(* Logix 5000 project; controller cow Emulate 5570 rev 36.11; software revision 36.00 *)

TASK MainTask (continuous, watchdog 500 ms) : MainProgram, Recipe, LED_UDP

MODULES
   Local : Emulate 5570 (ICP 0, rev 36.11)
      EN2T : 1756-EN2T (ICP 1, rev 12.1)
         Cow : 1756-ENBT (Ethernet 192.168.1.1, rev 5.1, Output RPI 10 ms)
            Caw1 : vendor 1 type 0 code 15 (ICP 0, rev 1.1, Output RPI 20 ms)
END_MODULES

TYPE ActLog :
STRUCT
   Time : DINT;
   STS : INT;
END_STRUCT
END_TYPE

TYPE Batch :
STRUCT
   Clear_Data : BOOL;
   LL : BOOL;
   Report_Log : BOOL;
   Value : INT;
   Batch : INT;
   Fall : INT;
   Target : INT;
   Net_Gross : DINT;
   Report : DINT[7];
   Scale : SCALE_WEIGHT;
   BinLog : BinLog[20];
END_STRUCT
END_TYPE

TYPE BinLog :
STRUCT
   SourceBin : INT;
   DestBin : INT;
   SetWeight : INT;
   StartTime : DINT;
   StopTime : DINT;
   pNumber : DINT;
   pNumberS : DINT[2];
END_STRUCT
END_TYPE

TYPE DateTime_Type :
STRUCT
   Year : DINT;
   Month : DINT;
   Day : DINT;
   Hour : DINT;
   Minute : DINT;
   Second : DINT;
   Microseconds : DINT;
END_STRUCT
END_TYPE

TYPE Part_Manual_Type :
STRUCT
   Bin : INT[5];
   Number : DINT[10];
   SetWeight : REAL[5];
   RealWeight : REAL[5];
   ErrorWeight : REAL[5];
END_STRUCT
END_TYPE

TYPE Part_Type :
STRUCT
   Bin : INT[20];
   Bin_Index : INT[20];
   Number : DINT[20];
   SetWeight : REAL[20];
   RealWeight : REAL[20];
   ErrorWeight : REAL[20];
END_STRUCT
END_TYPE

TYPE Part_Type_Hand :
STRUCT
   Number : DINT[30];
   SetWeight : REAL[30];
   RealWeight : REAL[30];
   ErrorWeight : REAL[30];
END_STRUCT
END_TYPE

TYPE Recipe_Type :
STRUCT
   Number : DINT[3];
   Desc : DINT[8];
   BatchSet : DINT;
   Date : DINT;
   pNumber : DINT[20];
   pSetWeight : REAL[20];
END_STRUCT
END_TYPE

TYPE REQUEST_PARAMETERS :
STRUCT
   Type : DINT;
   Addr : SockAddr;
END_STRUCT
END_TYPE

TYPE ScheduleLog :
STRUCT
   Number : DINT[3];
   StartTime : DINT;
   Batch : DINT;
END_STRUCT
END_TYPE

TYPE SockAddr :
STRUCT
   Family : INT;
   Port : INT;
   Addr : DINT;
END_STRUCT
END_TYPE

TYPE STR_OUT :
STRUCT
   LEN : DINT;
   BUFF : SINT[480];
END_STRUCT
END_TYPE

TYPE String20 :
STRUCT
   LEN : DINT;
   DATA : SINT[20];
END_STRUCT
END_TYPE

TYPE Sys_Data :
STRUCT
   MC : BOOL;
   AUTO_START : BOOL;
   AUTO_STOP : BOOL;
   EM : BOOL;
   AUTO : BOOL;
   MANUAL : BOOL;
   SIMULATE : BOOL;
   Monitor_PLC5 : BOOL;
   FlashFast : BOOL;
   FlashSlow : BOOL;
   Err_Reset : BOOL;
   PB : BOOL;
   Power : BOOL;
   Auto_Start_Enable : BOOL;
   Change_Bin_Ack : BOOL;
   FA : BOOL;
   Bin_Num_OK : BOOL;
   ClearLog : BOOL;
   Flag : BOOL;
   Alarm : BOOL;
   Compare_Bin : BOOL;
   OK : BOOL;
   BinLogStart : BOOL;
   Report_Log : BOOL;
   DropStop : BOOL;
   DM : BOOL;
   DropTimeS : INT;
   DropTime : TON_Second;
   BIN_SEL : INT;
   BIN_PLC : INT;
   BIN_SEL1 : INT;
   BinS_SEL1 : INT;
   BinS_SEL : INT;
   Day : INT;
   Day_Hour : INT;
   Year : INT;
   START_ACC : INT;
   Stop_ACC : INT;
   SEL_BIN : INT;
   MSG_ID : INT;
   MMDDHHMMS : DINT;
   sNumber : DINT;
   pNumber : DINT;
   NumberS : DINT[2];
   NumberSel : DINT[2];
   ActLog : ActLog[20];
   ChangeBin : TON_Second;
   StartT : TON_Second;
   StopT : TON_Second;
   TimeSet : TON_Second;
   SeqStartT : INT[21];
   SeqStopT : INT[21];
   BinLog : BinLog[20];
   SEL_Weight : REAL;
   Report : DINT[7];
END_STRUCT
END_TYPE

TYPE System_Common :
STRUCT
   Simulate : BOOL;
   Monitor_PLC5 : BOOL;
   FlashFast : BOOL;
   FlashSlow : BOOL;
   SY_PW_OK : BOOL;
   Err_Reset : BOOL;
   ClearLog : BOOL;
   PSH : BOOL;
   PSL : BOOL;
   Air_CLEAR : BOOL;
   DAY : INT;
   Day_Hour : INT;
   Year : INT;
   MMDDHHMMs : DINT;
END_STRUCT
END_TYPE

TYPE WRT_DATA :
STRUCT
   Timeout : DINT;
   ToAddr : SockAddr;
   Buffer : STR_OUT;
END_STRUCT
END_TYPE

ADD_ON_INSTRUCTION Air_Hammer   (* revision 1.0 *)
// 氣槌
VAR_INPUT
   PBM : BOOL; {visible}   // On/Off開關
   PB : BOOL;
   AB : BOOL;
   TH : BOOL;
END_VAR
VAR_OUTPUT
   SV : BOOL; {access Read Only, visible}   // 運轉
   MC : BOOL; {access Read Only}
   GL : BOOL; {access Read Only, visible}   // 運轉指示
END_VAR
VAR_INPUT
   Auto_on : BOOL; {visible}   // 連續
END_VAR
VAR_OUTPUT
   MotorType : BOOL; {visible}
END_VAR
VAR_IN_OUT
   Sys : Sys_Data; {required}   // 系統設定
END_VAR
VAR
   ONS : DINT; {access None}
   On_Time : TIMER := (PRE := 2000); {access None}
   Repeat_T : TIMER := (PRE := 2000); {access None}
END_VAR

ROUTINE Logic   (* ladder *)
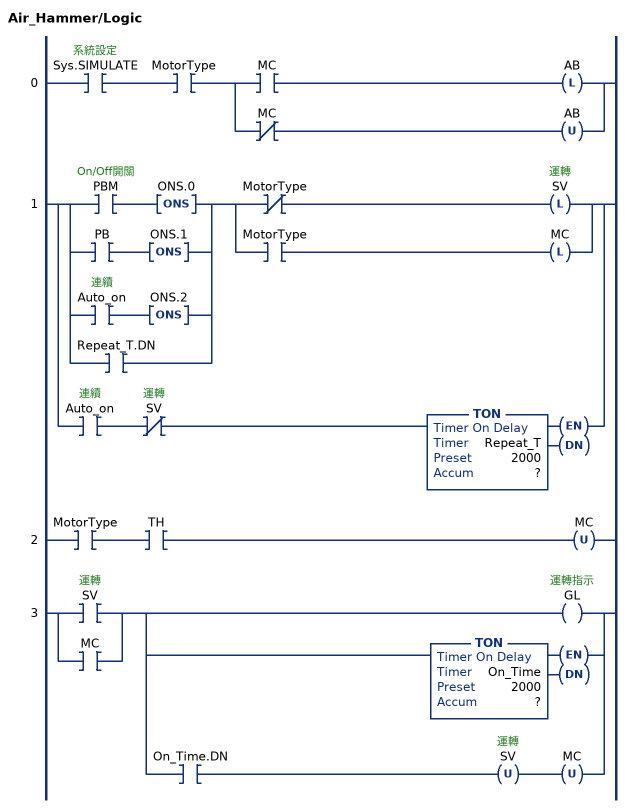
   0: XIC(Sys.SIMULATE)XIC(MotorType)[XIC(MC) OTL(AB) ,XIO(MC) OTU(AB) ];
   1: [[XIC(PBM) ONS(ONS.0) ,XIC(PB) ONS(ONS.1) ,XIC(Auto_on) ONS(ONS.2) ,XIC(Repeat_T.DN) ] [XIO(MotorType) OTL(SV) ,XIC(MotorType) OTL(MC) ] ,XIC(Auto_on) XIO(SV) TON(Repeat_T,?,?) ];
   2: XIC(MotorType)XIC(TH)OTU(MC);
   3: [XIC(SV) ,XIC(MC) ][OTE(GL) ,TON(On_Time,?,?) ,XIC(On_Time.DN) OTU(SV) OTU(MC) ];
END_ROUTINE
END_ADD_ON_INSTRUCTION

ADD_ON_INSTRUCTION Bin_Raw   (* revision 1.0 *)
VAR_OUTPUT
   HL : BOOL; {visible}
   LL : BOOL; {visible}
   FA : BOOL; {access Read Only, visible}
   Bin_sel : BOOL;
   Bin_Sel_OK : BOOL; {access Read Only}
   BIN_SELECTED : BOOL; {access Read Only}
   BIN_SELECTED1 : BOOL; {access Read Only}
   YL : BOOL; {access Read Only, visible}
   SV : BOOL;
END_VAR
VAR_INPUT
   LSO : BOOL;
END_VAR
VAR_OUTPUT
   CMD : BOOL; {visible}
   HGL : BOOL; {access Read Only, visible}
END_VAR
VAR_INPUT
   LS : BOOL; {access Read Only, visible}
   Change_Bin_Ack : BOOL;
   Bin_sel_No : BOOL;
END_VAR
VAR_OUTPUT
   HiSpeed : BOOL; {visible}
   LowSpeed : BOOL; {visible}
   DM : BOOL; {access Read Only, visible}
   SV_ON : BOOL;
   Disable : BOOL; {visible}
END_VAR
VAR_INPUT
   PB : BOOL;
END_VAR
VAR_OUTPUT
   GL : BOOL;
   Local_Sel : BOOL;
END_VAR
VAR_INPUT
   Bin : INT; {visible}
   Bin_ID : INT; {access Read Only, visible}
   Fall : REAL; {visible}
   Hi_Speed : INT := 80; {visible}
   Low_Speed : INT := 20; {visible}
   Low_Weight : INT := 5; {visible}
   Number : DINT; {visible}
   N0 : ALIAS FOR NumberS[0]; {visible}
   N1 : ALIAS FOR NumberS[1]; {visible}
END_VAR
VAR_IN_OUT
   Sys : Sys_Data; {required}
END_VAR
VAR
   Timer : TIMER := (PRE := 4000); {access None}
   ons : DINT; {access None}
   LVH_DELAY : TIMER := (PRE := 2000); {access None}
   NumberS : DINT[2];
END_VAR

ROUTINE Logic   (* ladder *)
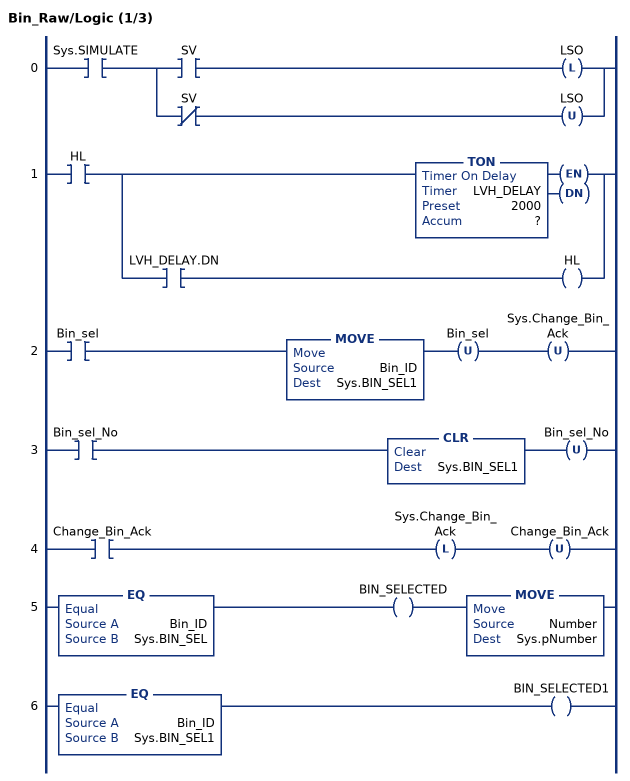
   0: XIC(Sys.SIMULATE)[XIC(SV) OTL(LSO) ,XIO(SV) OTU(LSO) ];
   1: XIC(HL)[TON(LVH_DELAY,?,?) ,XIC(LVH_DELAY.DN) OTE(HL) ];
   2: XIC(Bin_sel)MOVE(Bin_ID,Sys.BIN_SEL1)OTU(Bin_sel)OTU(Sys.Change_Bin_Ack);
   3: XIC(Bin_sel_No)CLR(Sys.BIN_SEL1)OTU(Bin_sel_No);
   4: XIC(Change_Bin_Ack)OTL(Sys.Change_Bin_Ack)OTU(Change_Bin_Ack);
   5: EQ(Bin_ID,Sys.BIN_SEL)OTE(BIN_SELECTED)MOVE(Number,Sys.pNumber);
   6: EQ(Bin_ID,Sys.BIN_SEL1)OTE(BIN_SELECTED1);
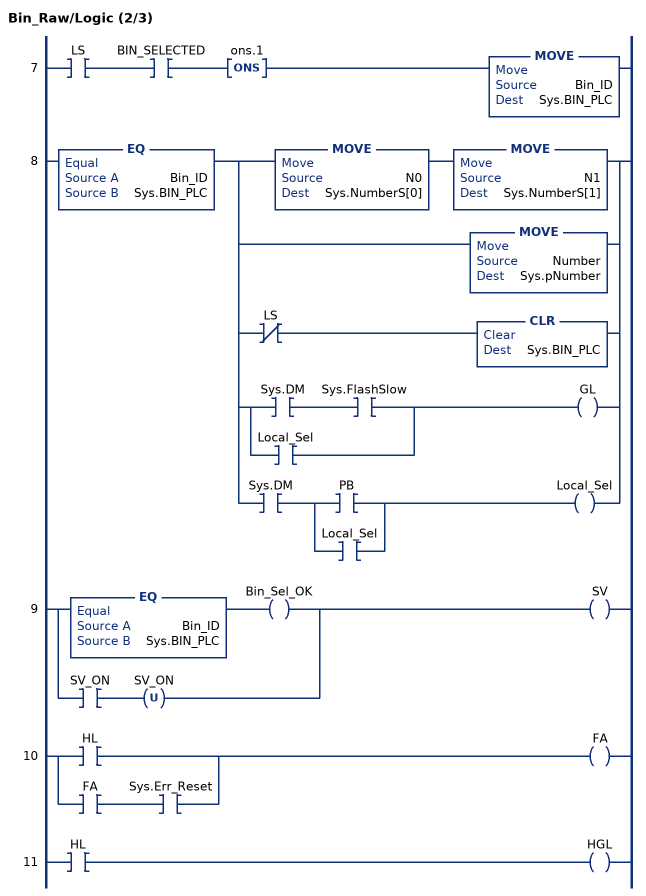
   7: XIC(LS)XIC(BIN_SELECTED)ONS(ons.1)MOVE(Bin_ID,Sys.BIN_PLC);
   8: EQ(Bin_ID,Sys.BIN_PLC)[MOVE(N0,Sys.NumberS[0]) MOVE(N1,Sys.NumberS[1]) ,MOVE(Number,Sys.pNumber) ,XIO(LS) CLR(Sys.BIN_PLC) ,[XIC(Sys.DM) XIC(Sys.FlashSlow) ,XIC(Local_Sel) ] OTE(GL) ,XIC(Sys.DM) [XIC(PB) ,XIC(Local_Sel) ] OTE(Local_Sel) ];
   9: [EQ(Bin_ID,Sys.BIN_PLC) OTE(Bin_Sel_OK) ,XIC(SV_ON) OTU(SV_ON) ]OTE(SV);
   10: [XIC(HL) ,XIC(FA) XIC(Sys.Err_Reset) ]OTE(FA);
   11: XIC(HL)OTE(HGL);
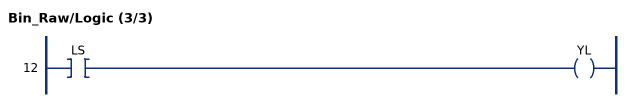
   12: XIC(LS)OTE(YL);
END_ROUTINE
END_ADD_ON_INSTRUCTION

ADD_ON_INSTRUCTION Branch_SV2   (* revision 1.0 *)
VAR_INPUT
   LSY : BOOL; {visible}
   LSX : BOOL; {visible}
END_VAR
VAR_OUTPUT
   SVX : BOOL; {access Read Only, visible}
   SVY : BOOL; {access Read Only, visible}
   FA : BOOL; {visible}
   GLX : BOOL; {access Read Only}
   GLY : BOOL; {access Read Only}
   Manual : BOOL;
   SVXPB : BOOL; {visible}
   SVYPB : BOOL; {visible}
   Auto : BOOL;
   Not_AOI_Control : BOOL; {visible}
END_VAR
VAR_INPUT
   InterLock : BOOL;
END_VAR
VAR_IN_OUT
   STS : INT; {required}
   Sys : Sys_Data; {required}
END_VAR
VAR
   SV : BOOL; {access None}
   ONS : DINT; {access None}
   DELAY : TIMER := (PRE := 3000); {access None}
   ActLog : ActLog[20];
   LastOnTime : DINT;
   LastOffTime : DINT;
END_VAR

ROUTINE Logic   (* ladder *)
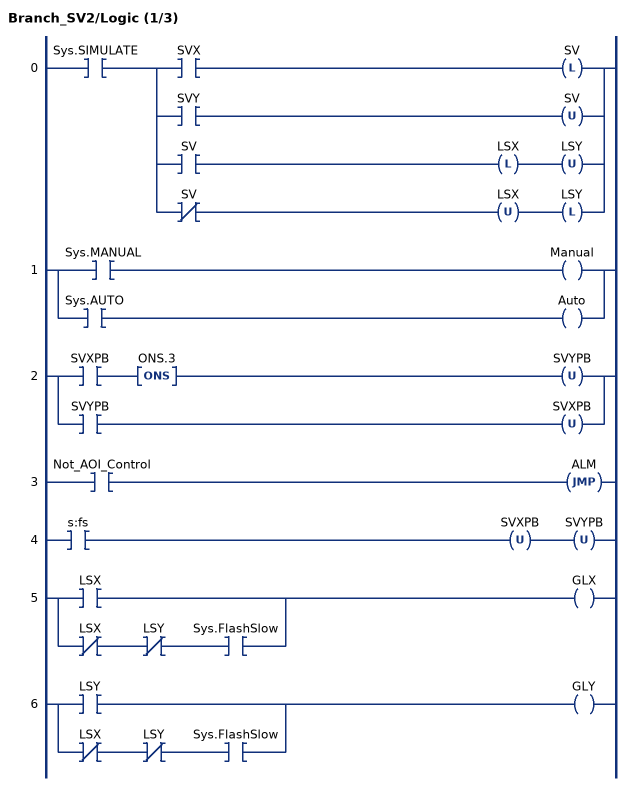
   0: XIC(Sys.SIMULATE)[XIC(SVX) OTL(SV) ,XIC(SVY) OTU(SV) ,XIC(SV) OTL(LSX) OTU(LSY) ,XIO(SV) OTU(LSX) OTL(LSY) ];
   1: [XIC(Sys.MANUAL) OTE(Manual) ,XIC(Sys.AUTO) OTE(Auto) ];
   2: [XIC(SVXPB) ONS(ONS.3) OTU(SVYPB) ,XIC(SVYPB) OTU(SVXPB) ];
   3: XIC(Not_AOI_Control)JMP(ALM);
   4: XIC(s:fs)OTU(SVXPB)OTU(SVYPB);
   5: [XIC(LSX) ,XIO(LSX) XIO(LSY) XIC(Sys.FlashSlow) ]OTE(GLX);
   6: [XIC(LSY) ,XIO(LSX) XIO(LSY) XIC(Sys.FlashSlow) ]OTE(GLY);
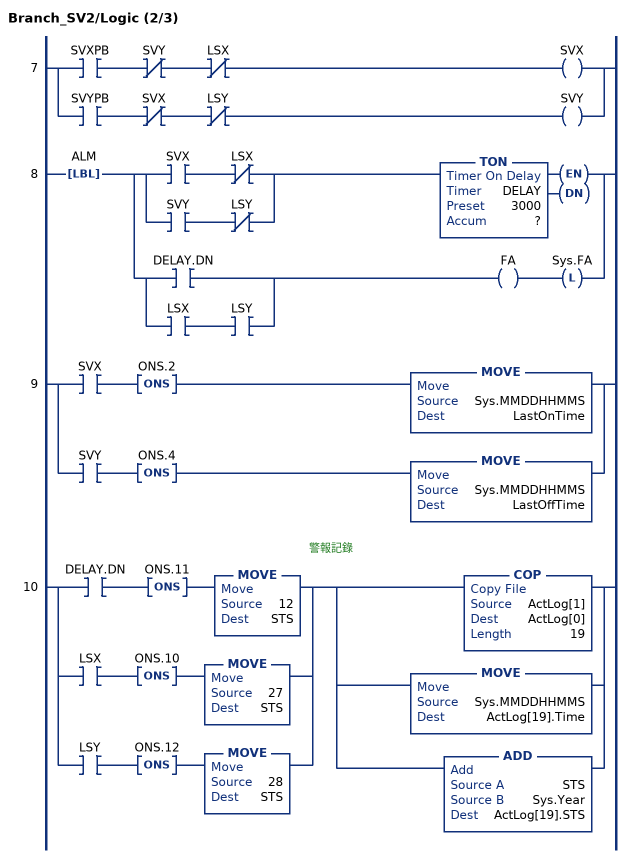
   7: [XIC(SVXPB) XIO(SVY) XIO(LSX) OTE(SVX) ,XIC(SVYPB) XIO(SVX) XIO(LSY) OTE(SVY) ];
   8: LBL(ALM)[[XIC(SVX) XIO(LSX) ,XIC(SVY) XIO(LSY) ] TON(DELAY,?,?) ,[XIC(DELAY.DN) ,XIC(LSX) XIC(LSY) ] OTE(FA) OTL(Sys.FA) ];
   9: [XIC(SVX) ONS(ONS.2) MOVE(Sys.MMDDHHMMS,LastOnTime) ,XIC(SVY) ONS(ONS.4) MOVE(Sys.MMDDHHMMS,LastOffTime) ];
   // 警報記錄
   10: [XIC(DELAY.DN) ONS(ONS.11) MOVE(12,STS) ,[XIC(LSX) ONS(ONS.10) MOVE(27,STS) ,XIC(LSY) ONS(ONS.12) MOVE(28,STS) ] ][COP(ActLog[1],ActLog[0],19) ,MOVE(Sys.MMDDHHMMS,ActLog[19].Time) ,ADD(STS,Sys.Year,ActLog[19].STS) ];
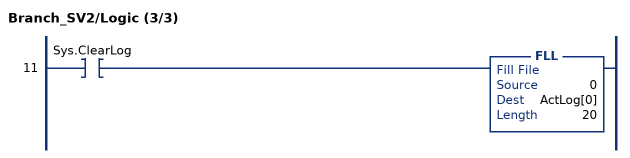
   11: XIC(Sys.ClearLog)FLL(0,ActLog[0],20);
END_ROUTINE
END_ADD_ON_INSTRUCTION

ADD_ON_INSTRUCTION DateTime_String   (* revision 1.0 *)
VAR_IN_OUT
   Now : DateTime_Type; {required}
   DateTimes : STRING; {required}
END_VAR
VAR
   HOUR : STRING; {access None}
   MINUTE : STRING; {access None}
   SECOND : STRING; {access None}
   zero : STRING := '0'; {access None}
   COLN : STRING := ':'; {access None}
   Prev_Second : DINT; {access None}
   Day : STRING; {access None}
   Month : STRING; {access None}
   Year : STRING; {access None}
   Da : STRING := '/'; {access None}
   Blank : STRING := '  '; {access None}
END_VAR

ROUTINE Logic   (* ladder *)
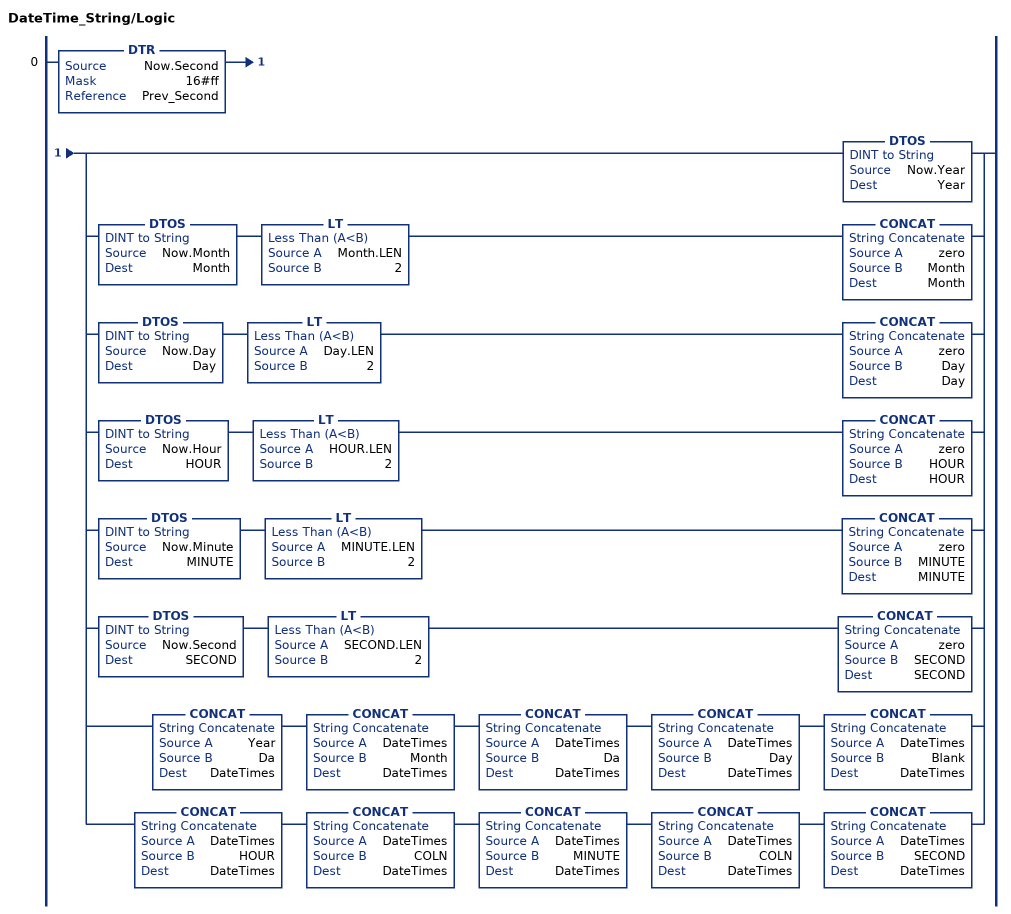
   0: DTR(Now.Second,16#ff,Prev_Second)[DTOS(Now.Year,Year) ,DTOS(Now.Month,Month) LT(Month.LEN,2) CONCAT(zero,Month,Month) ,DTOS(Now.Day,Day) LT(Day.LEN,2) CONCAT(zero,Day,Day) ,DTOS(Now.Hour,HOUR) LT(HOUR.LEN,2) CONCAT(zero,HOUR,HOUR) ,DTOS(Now.Minute,MINUTE) LT(MINUTE.LEN,2) CONCAT(zero,MINUTE,MINUTE) ,DTOS(Now.Second,SECOND) LT(SECOND.LEN,2) CONCAT(zero,SECOND,SECOND) ,CONCAT(Year,Da,DateTimes) CONCAT(DateTimes,Month,DateTimes) CONCAT(DateTimes,Da,DateTimes) CONCAT(DateTimes,Day,DateTimes) CONCAT(DateTimes,Blank,DateTimes) ,CONCAT(DateTimes,HOUR,DateTimes) CONCAT(DateTimes,COLN,DateTimes) CONCAT(DateTimes,MINUTE,DateTimes) CONCAT(DateTimes,COLN,DateTimes) CONCAT(DateTimes,SECOND,DateTimes) ];
END_ROUTINE
END_ADD_ON_INSTRUCTION

ADD_ON_INSTRUCTION Divider   (* revision 1.0 *)
VAR_INPUT
   AB : BOOL; {visible}
END_VAR
VAR_OUTPUT
   MC : BOOL; {access Read Only, visible}
END_VAR
VAR_INPUT
   TH : BOOL; {visible}
END_VAR
VAR_OUTPUT
   FA : BOOL; {visible}
END_VAR
VAR_INPUT
   MANUAL_ON : BOOL; {visible}
   AUTO_ON : BOOL;
END_VAR
VAR_OUTPUT
   MANUAL : BOOL; {visible}
   OverTime : BOOL; {visible}
   LS1 : ALIAS FOR LS.1;
   LS2 : ALIAS FOR LS.2;
   LS3 : ALIAS FOR LS.3;
   LS4 : ALIAS FOR LS.4;
   LS5 : ALIAS FOR LS.5;
   LS6 : ALIAS FOR LS.6;
   LS7 : ALIAS FOR LS.7;
   LS8 : ALIAS FOR LS.8;
   LS9 : ALIAS FOR LS.9;
   LS10 : ALIAS FOR LS.10;
   LS11 : ALIAS FOR LS.11;
   LS12 : ALIAS FOR LS.12;
   LS_ON : BOOL;
   Not_AOI_Control : BOOL; {visible}
   Bin_select : BOOL; {visible}
   Simulate : ALIAS FOR Simulate_POS.ACC; {access Read Only}
END_VAR
VAR_IN_OUT
   STS : INT; {required}
   Sys : Sys_Data; {required}
END_VAR
VAR
   DELAY : TIMER := (PRE := 1000); {access None}
   Simulate_TIMER : TIMER := (PRE := 1000); {access None}
   Simulate_POS : COUNTER := (PRE := 7); {access Read Only}
   ONS : DINT; {access None}
   error_delay : TIMER := (PRE := 5000); {access None}
   MC_RUN_T : TIMER := (PRE := 40000); {access None}
   LS : DINT;
   ActLog : ActLog[20];
   LastOnTime : DINT;
   LastOffTime : DINT;
END_VAR

ROUTINE Logic   (* ladder *)
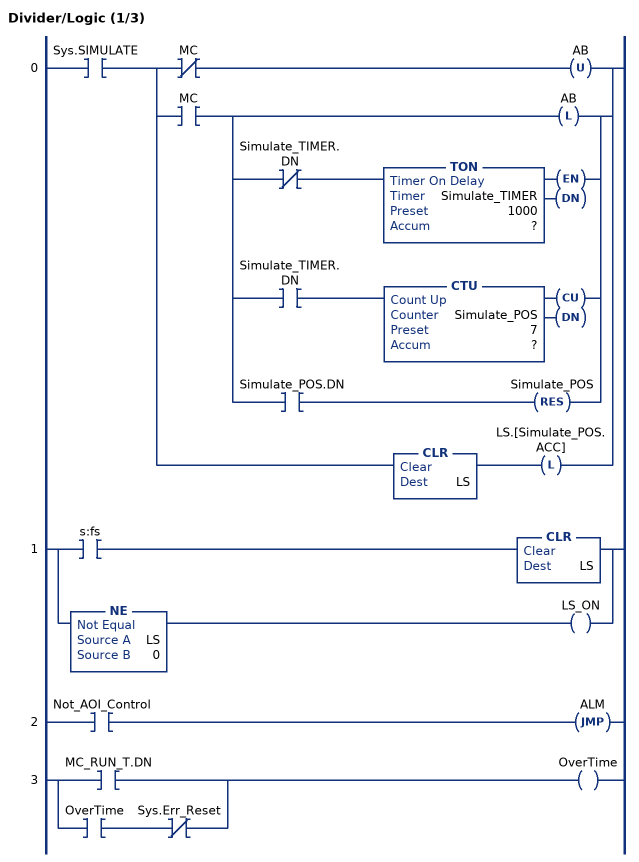
   0: XIC(Sys.SIMULATE)[XIO(MC) OTU(AB) ,XIC(MC) [OTL(AB) ,XIO(Simulate_TIMER.DN) TON(Simulate_TIMER,?,?) ,XIC(Simulate_TIMER.DN) CTU(Simulate_POS,?,?) ,XIC(Simulate_POS.DN) RES(Simulate_POS) ] ,CLR(LS) OTL(LS.[Simulate_POS.ACC]) ];
   1: [XIC(s:fs) CLR(LS) ,NE(LS,0) OTE(LS_ON) ];
   2: XIC(Not_AOI_Control)JMP(ALM);
   3: [XIC(MC_RUN_T.DN) ,XIC(OverTime) XIO(Sys.Err_Reset) ]OTE(OverTime);
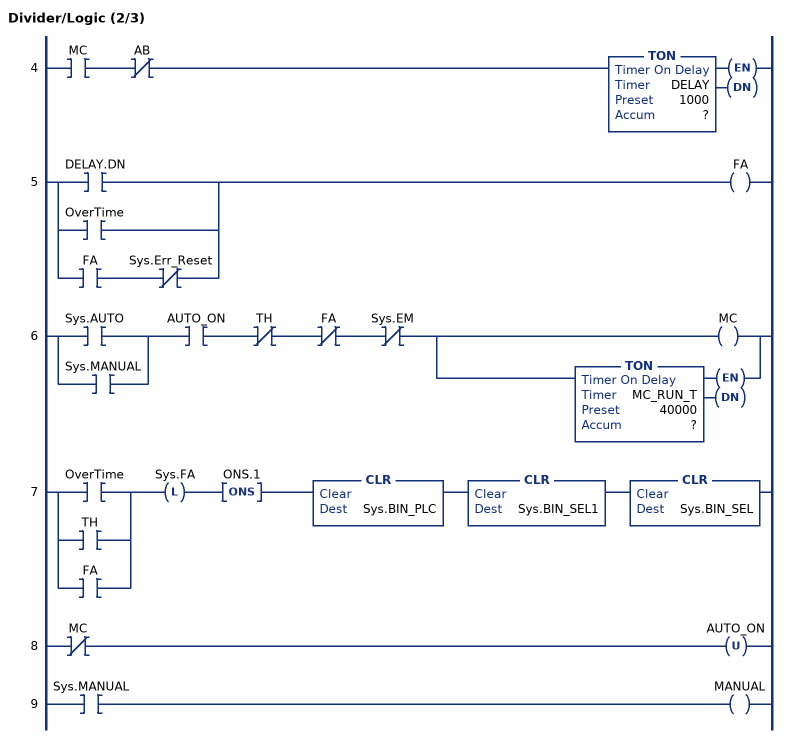
   4: XIC(MC)XIO(AB)TON(DELAY,?,?);
   5: [XIC(DELAY.DN) ,XIC(OverTime) ,XIC(FA) XIO(Sys.Err_Reset) ]OTE(FA);
   6: [XIC(Sys.AUTO) ,XIC(Sys.MANUAL) ]XIC(AUTO_ON)XIO(TH)XIO(FA)XIO(Sys.EM)[OTE(MC) ,TON(MC_RUN_T,?,?) ];
   7: [XIC(OverTime) ,XIC(TH) ,XIC(FA) ]OTL(Sys.FA)ONS(ONS.1)CLR(Sys.BIN_PLC)CLR(Sys.BIN_SEL1)CLR(Sys.BIN_SEL);
   8: XIO(MC)OTU(AUTO_ON);
   9: XIC(Sys.MANUAL)OTE(MANUAL);
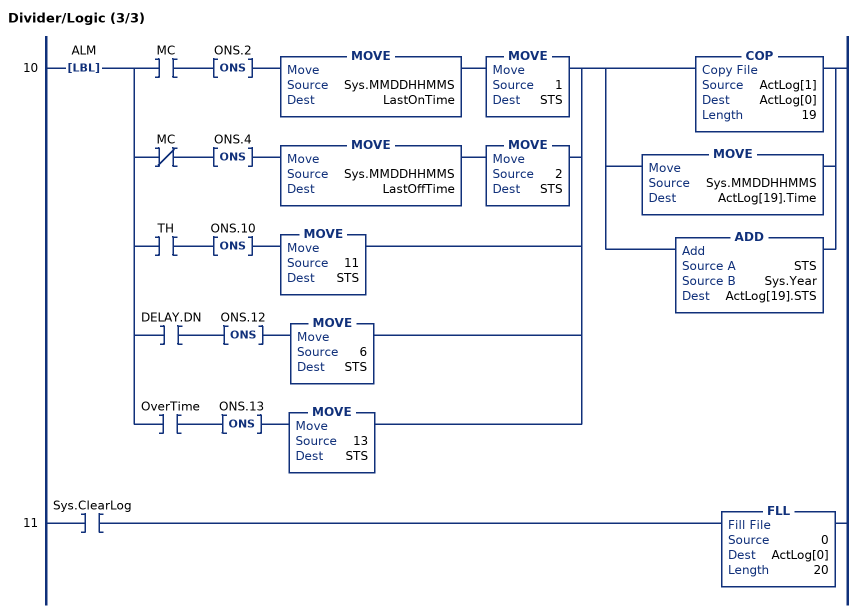
   10: LBL(ALM)[XIC(MC) ONS(ONS.2) MOVE(Sys.MMDDHHMMS,LastOnTime) MOVE(1,STS) ,XIO(MC) ONS(ONS.4) MOVE(Sys.MMDDHHMMS,LastOffTime) MOVE(2,STS) ,XIC(TH) ONS(ONS.10) MOVE(11,STS) ,XIC(DELAY.DN) ONS(ONS.12) MOVE(6,STS) ,XIC(OverTime) ONS(ONS.13) MOVE(13,STS) ][COP(ActLog[1],ActLog[0],19) ,MOVE(Sys.MMDDHHMMS,ActLog[19].Time) ,ADD(STS,Sys.Year,ActLog[19].STS) ];
   11: XIC(Sys.ClearLog)FLL(0,ActLog[0],20);
END_ROUTINE
END_ADD_ON_INSTRUCTION

ADD_ON_INSTRUCTION Gate   (* revision 1.0 *)
VAR_INPUT
   LSO : BOOL; {visible}
   LSK : BOOL; {visible}
END_VAR
VAR_OUTPUT
   SV : BOOL; {visible}
   Auto_On : BOOL;
   Manual : BOOL; {visible}
   FA : BOOL; {visible}
   OPEN : BOOL; {visible}
   InterLock : BOOL; {access Read Only, visible}
   Auto : BOOL;
   PB : BOOL;
   GL : BOOL; {access Read Only, visible}
END_VAR
VAR_INPUT
   LL : BOOL;
END_VAR
VAR_OUTPUT
   Not_AOI_Control : BOOL; {visible}
   Lock : BOOL;
   LSO_Delay : BOOL;
   Off_Delay : BOOL;
END_VAR
VAR_IN_OUT
   STS : INT; {required}
   Sys : Sys_Data; {required}
END_VAR
VAR
   Open_Delay : TIMER := (PRE := 500); {access None}
   Close_Delay : TIMER := (PRE := 500); {access None}
   TimeOut : TIMER := (PRE := 3000); {access None}
   Interlock_Delay : TIMER := (PRE := 500); {access None}
   ActLog : ActLog[20];
   ONS : DINT; {access None}
   LS_Delay : TIMER[2] := ([0].PRE := 1000, [1].PRE := 1000); {access None}
   PB_Delay : TIMER := (PRE := 500); {access None}
   LSO_DelayT : TIMER := (PRE := 2000); {access None}
   off_DelayT : TIMER := (PRE := 2000); {access None}
END_VAR

ROUTINE Logic   (* ladder *)
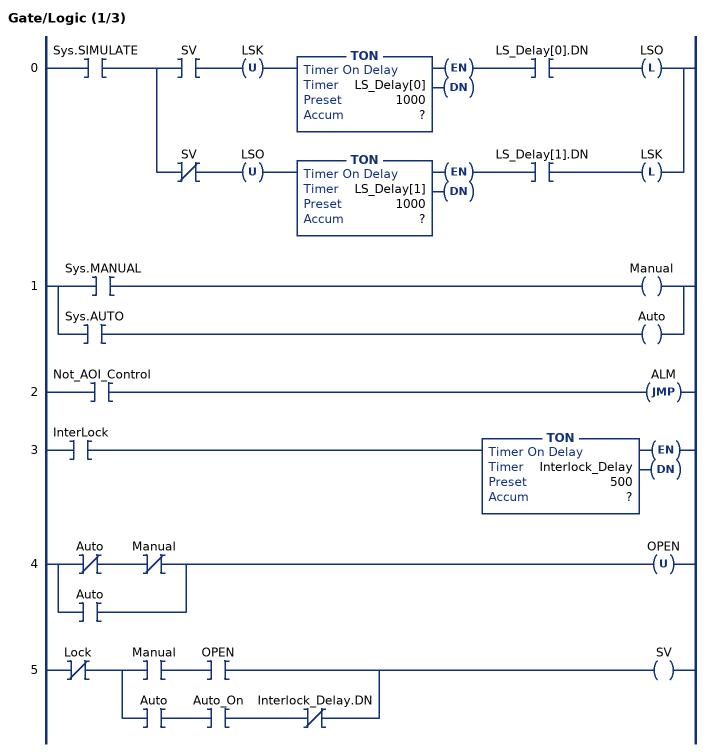
   0: XIC(Sys.SIMULATE)[XIC(SV) OTU(LSK) TON(LS_Delay[0],?,?) XIC(LS_Delay[0].DN) OTL(LSO) ,XIO(SV) OTU(LSO) TON(LS_Delay[1],?,?) XIC(LS_Delay[1].DN) OTL(LSK) ];
   1: [XIC(Sys.MANUAL) OTE(Manual) ,XIC(Sys.AUTO) OTE(Auto) ];
   2: XIC(Not_AOI_Control)JMP(ALM);
   3: XIC(InterLock)TON(Interlock_Delay,?,?);
   4: [XIO(Auto) XIO(Manual) ,XIC(Auto) ]OTU(OPEN);
   5: XIO(Lock)[XIC(Manual) XIC(OPEN) ,XIC(Auto) XIC(Auto_On) XIO(Interlock_Delay.DN) ]OTE(SV);
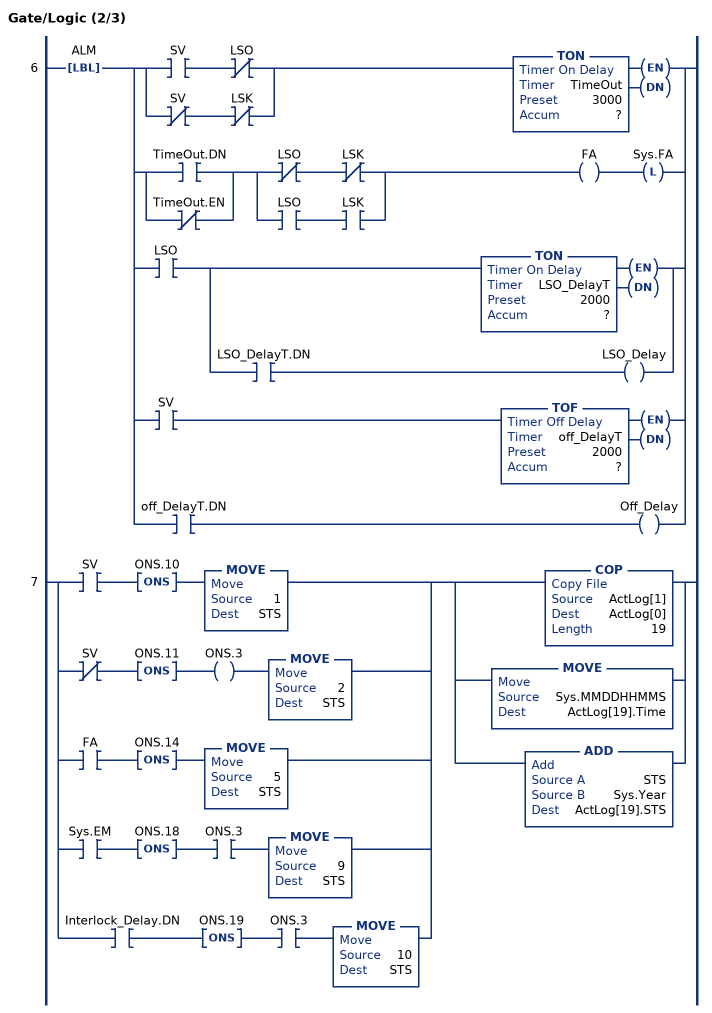
   6: LBL(ALM)[[XIC(SV) XIO(LSO) ,XIO(SV) XIO(LSK) ] TON(TimeOut,?,?) ,[XIC(TimeOut.DN) ,XIO(TimeOut.EN) ] [XIO(LSO) XIO(LSK) ,XIC(LSO) XIC(LSK) ] OTE(FA) OTL(Sys.FA) ,XIC(LSO) [TON(LSO_DelayT,?,?) ,XIC(LSO_DelayT.DN) OTE(LSO_Delay) ] ,XIC(SV) TOF(off_DelayT,?,?) ,XIC(off_DelayT.DN) OTE(Off_Delay) ];
   7: [[XIC(SV) ONS(ONS.10) MOVE(1,STS) ,XIO(SV) ONS(ONS.11) OTE(ONS.3) MOVE(2,STS) ] ,XIC(FA) ONS(ONS.14) MOVE(5,STS) ,XIC(Sys.EM) ONS(ONS.18) XIC(ONS.3) MOVE(9,STS) ,XIC(Interlock_Delay.DN) ONS(ONS.19) XIC(ONS.3) MOVE(10,STS) ][COP(ActLog[1],ActLog[0],19) ,MOVE(Sys.MMDDHHMMS,ActLog[19].Time) ,ADD(STS,Sys.Year,ActLog[19].STS) ];
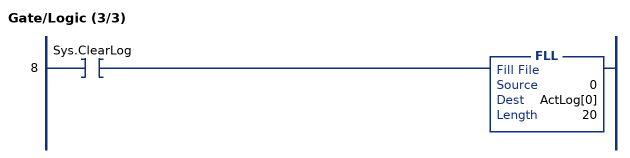
   8: XIC(Sys.ClearLog)FLL(0,ActLog[0],20);
END_ROUTINE
END_ADD_ON_INSTRUCTION

ADD_ON_INSTRUCTION Inverter   (* revision 1.0 *)
VAR_INPUT
   AB : BOOL; {visible}
END_VAR
VAR_OUTPUT
   MC : BOOL; {access Read Only, visible}
END_VAR
VAR_INPUT
   TH : BOOL; {visible}
END_VAR
VAR_OUTPUT
   RMC : BOOL; {visible}
   AUTO_ON : BOOL;
END_VAR
VAR_INPUT
   Manual_HZ : INT := 10; {visible}
   HZ : INT; {visible}
END_VAR
VAR_IN_OUT
   STS : INT; {required}
   Sys : Sys_Data; {required}
END_VAR
VAR
   DELAY : TIMER := (PRE := 100); {access None}
   ONS : DINT; {access None}
   AlmLog : DINT[6]; {access Read Only}
   ALM_ID : DINT; {access None}
   RunTIme : TIMER := (PRE := 99999); {access Read Only}
END_VAR

ROUTINE Logic   (* ladder *)
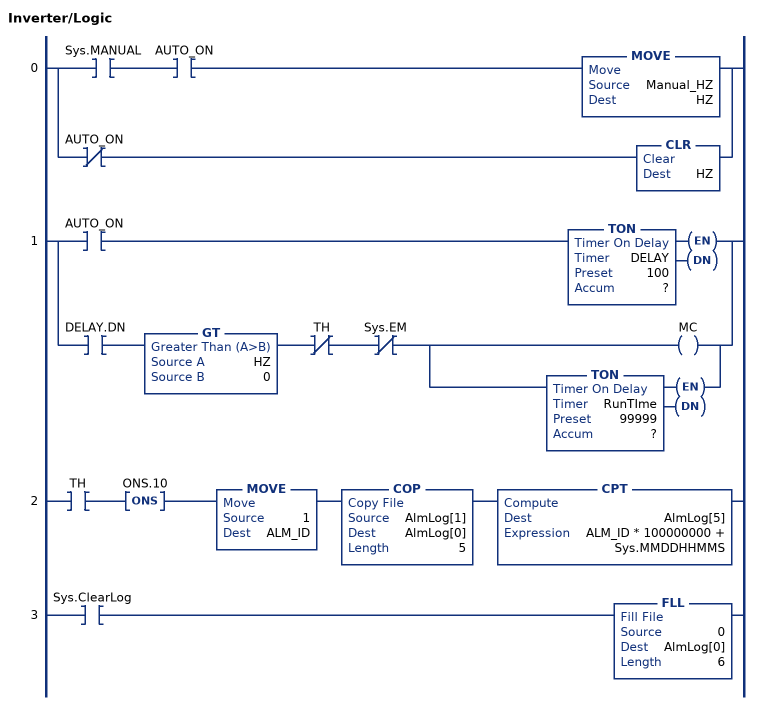
   0: [XIC(Sys.MANUAL) XIC(AUTO_ON) MOVE(Manual_HZ,HZ) ,XIO(AUTO_ON) CLR(HZ) ];
   1: [XIC(AUTO_ON) TON(DELAY,?,?) ,XIC(DELAY.DN) GT(HZ,0) XIO(TH) XIO(Sys.EM) [OTE(MC) ,TON(RunTIme,?,?) ] ];
   2: XIC(TH)ONS(ONS.10)MOVE(1,ALM_ID)COP(AlmLog[1],AlmLog[0],5)CPT(AlmLog[5],ALM_ID * 100000000 + Sys.MMDDHHMMS);
   3: XIC(Sys.ClearLog)FLL(0,AlmLog[0],6);
END_ROUTINE
END_ADD_ON_INSTRUCTION

ADD_ON_INSTRUCTION LED_CMD   (* revision 1.0 *)
VAR_IN_OUT
   strCMD : STRING; {required}
   strOut : STRING; {required}
END_VAR
VAR
   sum : SINT; {access None}
   index : DINT; {access None}
   strSum : STRING; {access None}
END_VAR

ROUTINE Logic   (* ladder *)
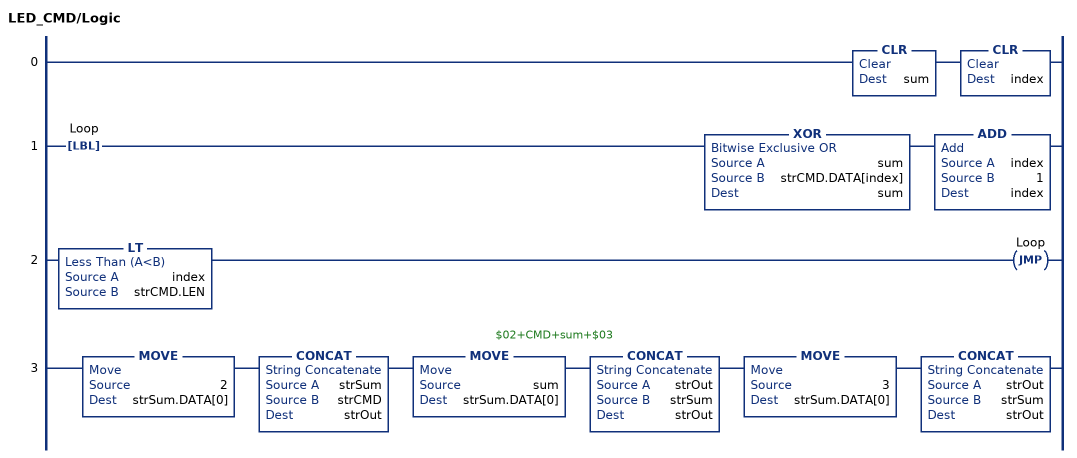
   0: CLR(sum)CLR(index);
   1: LBL(Loop)XOR(sum,strCMD.DATA[index],sum)ADD(index,1,index);
   2: LT(index,strCMD.LEN)JMP(Loop);
   // $02+CMD+sum+$03
   3: MOVE(2,strSum.DATA[0])CONCAT(strSum,strCMD,strOut)MOVE(sum,strSum.DATA[0])CONCAT(strOut,strSum,strOut)MOVE(3,strSum.DATA[0])CONCAT(strOut,strSum,strOut);
END_ROUTINE
END_ADD_ON_INSTRUCTION

ADD_ON_INSTRUCTION MotorX   (* revision 1.0 *)
VAR_INPUT
   AB : BOOL; {visible}
END_VAR
VAR_OUTPUT
   MC : BOOL; {access Read Only, visible}
END_VAR
VAR_INPUT
   TH : BOOL; {visible}
   PB : BOOL;
   PBM : BOOL;
END_VAR
VAR_OUTPUT
   GL : BOOL; {access Read Only, visible}
END_VAR
VAR_INPUT
   HL : BOOL;
   LL : BOOL;
END_VAR
VAR_OUTPUT
   HLGL : BOOL; {access Read Only}
   LLGL : BOOL; {access Read Only}
END_VAR
VAR_INPUT
   EM : BOOL; {visible}
   MANUAL_ON : BOOL;
   AUTO_ON : BOOL;
END_VAR
VAR_OUTPUT
   Manual : BOOL; {visible}
   Auto : BOOL;
   FA : BOOL; {visible}
   InterLock : BOOL; {visible}
END_VAR
VAR_INPUT
   AUTO_ON_OFF : BOOL;
   AB1 : BOOL;
   AB2 : BOOL;
   AB3 : BOOL;
END_VAR
VAR_OUTPUT
   MC1 : BOOL; {access Read Only}
   MC2 : BOOL; {access Read Only}
   MC3 : BOOL; {access Read Only}
END_VAR
VAR_INPUT
   SP : BOOL;
   AS : BOOL;
   JM : BOOL; {access Read Only}
END_VAR
VAR_OUTPUT
   DM : BOOL;
   SP_ALM : BOOL; {visible}
   MC_Type : BOOL;
END_VAR
VAR_INPUT
   Temp : BOOL;
END_VAR
VAR_OUTPUT
   SV : BOOL; {access Read Only}
END_VAR
VAR_INPUT
   LSO : BOOL;
END_VAR
VAR_OUTPUT
   LSK : BOOL;
END_VAR
VAR_INPUT
   PS : BOOL;
   Protect : BOOL;
END_VAR
VAR_OUTPUT
   SP_Check : BOOL; {visible}
   Not_AOI_Control : BOOL; {access Read Only}
   CLEAN : BOOL;
   CLEAN_Reset : BOOL;
   Group_On : BOOL;
END_VAR
VAR_INPUT
   Sel : BOOL;
END_VAR
VAR_OUTPUT
   Alarm : BOOL;
   Disable_SP_Alarm : BOOL;
   START_DN : BOOL;
   DMPB : BOOL;
END_VAR
VAR_INPUT
   AMP : REAL;
END_VAR
VAR_OUTPUT
   RPM : INT;
   ReStart : INT;
END_VAR
VAR_IN_OUT
   STS : INT; {required}
   Sys : Sys_Data; {required}
END_VAR
VAR
   START_T : TIMER := (PRE := 20000); {access None}
   DELAY : TIMER := (PRE := 3000); {access None}
   error_delay : TIMER := (PRE := 5000); {access None}
   ONS : DINT; {access None}
        .7   // auto_oper
        .8   // Manual_oper
   Interlock_delay : TIMER := (PRE := 1000); {access None}
   SP_Check_T : TIMER := (PRE := 6000); {access None}
   ReStart_T : TIMER := (PRE := 3000); {access None}
   JM_Delay : TIMER := (PRE := 2000); {access None}
   ActLog : ActLog[20];
   LastOnTime : DINT;
   LastOffTime : DINT;
END_VAR

ROUTINE Logic   (* ladder *)
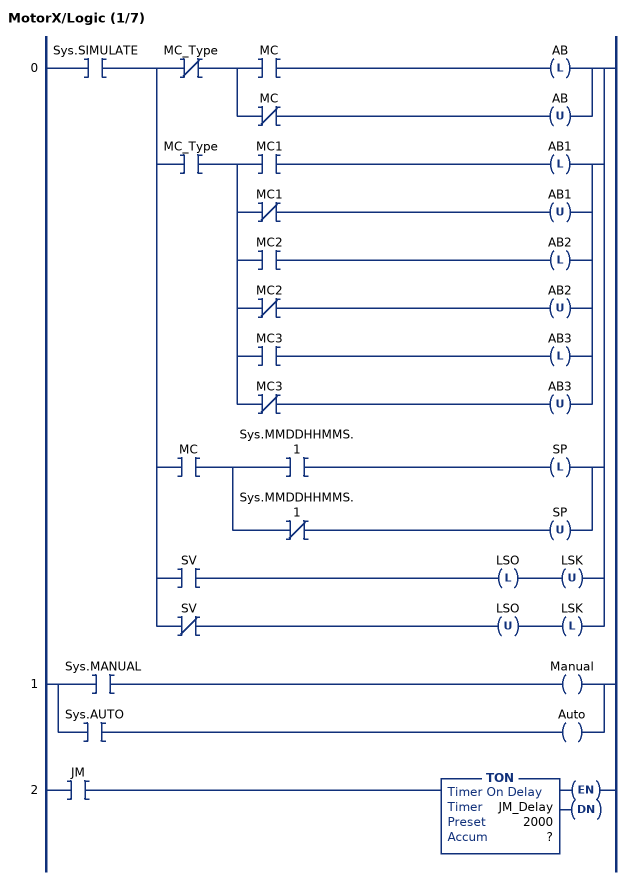
   0: XIC(Sys.SIMULATE)[XIO(MC_Type) [XIC(MC) OTL(AB) ,XIO(MC) OTU(AB) ] ,XIC(MC_Type) [XIC(MC1) OTL(AB1) ,XIO(MC1) OTU(AB1) ,XIC(MC2) OTL(AB2) ,XIO(MC2) OTU(AB2) ,XIC(MC3) OTL(AB3) ,XIO(MC3) OTU(AB3) ] ,XIC(MC) [XIC(Sys.MMDDHHMMS.1) OTL(SP) ,XIO(Sys.MMDDHHMMS.1) OTU(SP) ] ,[XIC(SV) OTL(LSO) OTU(LSK) ,XIO(SV) OTU(LSO) OTL(LSK) ] ];
   1: [XIC(Sys.MANUAL) OTE(Manual) ,XIC(Sys.AUTO) OTE(Auto) ];
   2: XIC(JM)TON(JM_Delay,?,?);
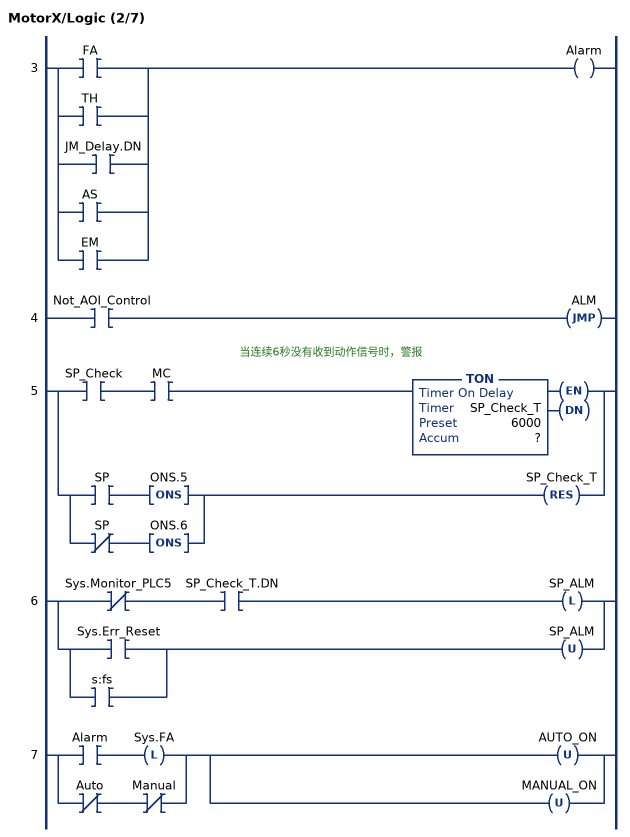
   3: [XIC(FA) ,XIC(TH) ,XIC(JM_Delay.DN) ,XIC(AS) ,XIC(EM) ]OTE(Alarm);
   4: XIC(Not_AOI_Control)JMP(ALM);
   // 当连续6秒没有收到动作信号时，警报
   5: [XIC(SP_Check) XIC(MC) TON(SP_Check_T,?,?) ,[XIC(SP) ONS(ONS.5) ,XIO(SP) ONS(ONS.6) ] RES(SP_Check_T) ];
   6: [XIO(Sys.Monitor_PLC5) XIC(SP_Check_T.DN) OTL(SP_ALM) ,[XIC(Sys.Err_Reset) ,XIC(s:fs) ] OTU(SP_ALM) ];
   7: [XIC(Alarm) OTL(Sys.FA) ,XIO(Auto) XIO(Manual) ][OTU(AUTO_ON) ,OTU(MANUAL_ON) ];
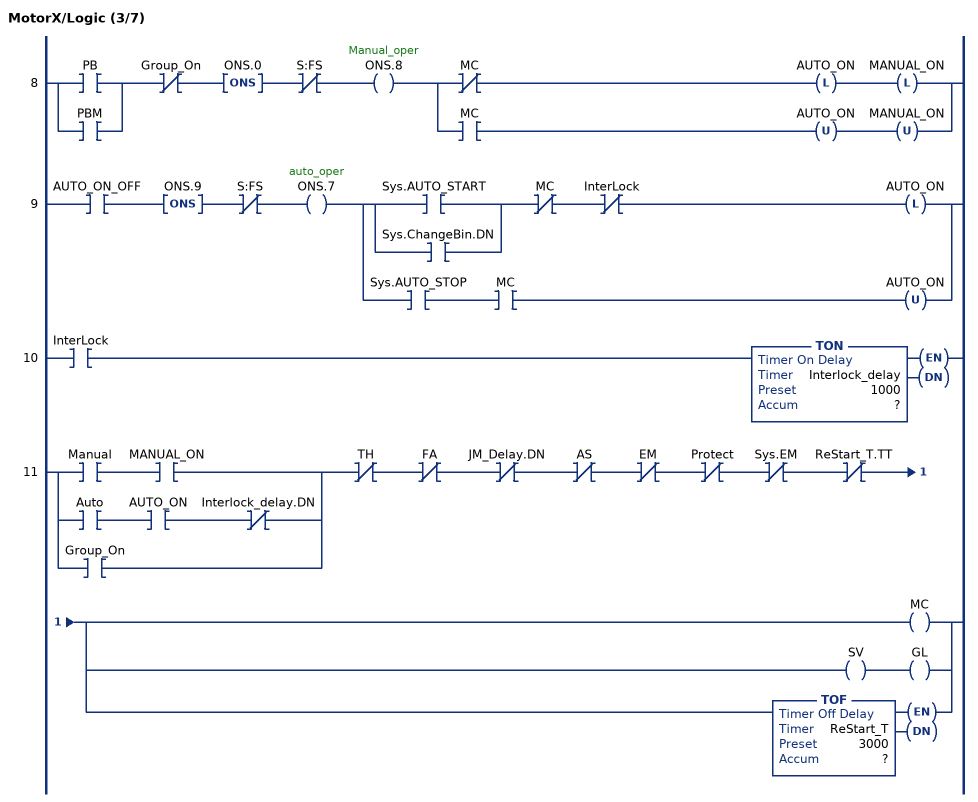
   8: [XIC(PB) ,XIC(PBM) ]XIO(Group_On)ONS(ONS.0)XIO(S:FS)OTE(ONS.8)[XIO(MC) OTL(AUTO_ON) OTL(MANUAL_ON) ,XIC(MC) OTU(AUTO_ON) OTU(MANUAL_ON) ];
   9: XIC(AUTO_ON_OFF)ONS(ONS.9)XIO(S:FS)OTE(ONS.7)[[XIC(Sys.AUTO_START) ,XIC(Sys.ChangeBin.DN) ] XIO(MC) XIO(InterLock) OTL(AUTO_ON) ,XIC(Sys.AUTO_STOP) XIC(MC) OTU(AUTO_ON) ];
   10: XIC(InterLock)TON(Interlock_delay,?,?);
   11: [XIC(Manual) XIC(MANUAL_ON) ,XIC(Auto) XIC(AUTO_ON) XIO(Interlock_delay.DN) ,XIC(Group_On) ]XIO(TH)XIO(FA)XIO(JM_Delay.DN)XIO(AS)XIO(EM)XIO(Protect)XIO(Sys.EM)XIO(ReStart_T.TT)[OTE(MC) ,OTE(SV) OTE(GL) ,TOF(ReStart_T,?,?) ];
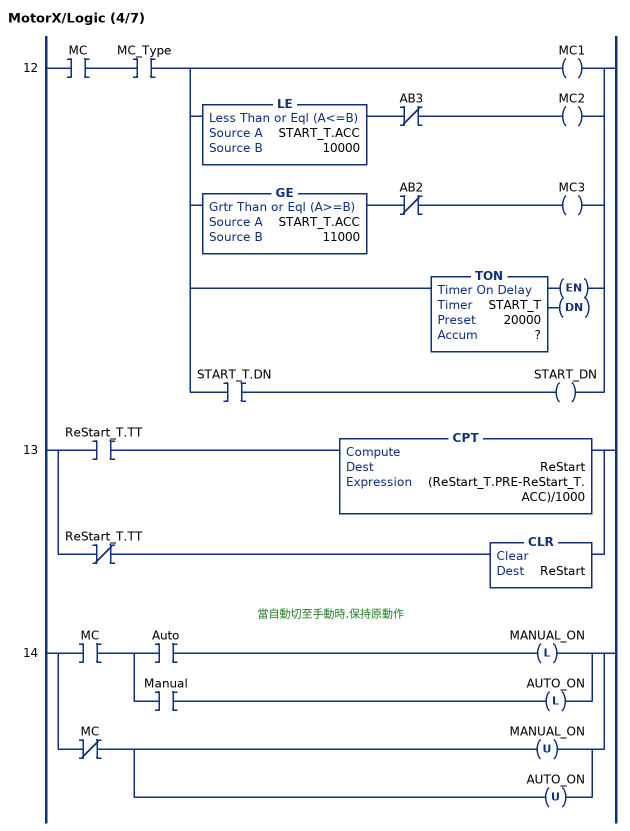
   12: XIC(MC)XIC(MC_Type)[OTE(MC1) ,LE(START_T.ACC,10000) XIO(AB3) OTE(MC2) ,GE(START_T.ACC,11000) XIO(AB2) OTE(MC3) ,TON(START_T,?,?) ,XIC(START_T.DN) OTE(START_DN) ];
   13: [XIC(ReStart_T.TT) CPT(ReStart,(ReStart_T.PRE-ReStart_T.ACC)/1000) ,XIO(ReStart_T.TT) CLR(ReStart) ];
   // 當自動切至手動時,保持原動作
   14: [XIC(MC) [XIC(Auto) OTL(MANUAL_ON) ,XIC(Manual) OTL(AUTO_ON) ] ,XIO(MC) [OTU(MANUAL_ON) ,OTU(AUTO_ON) ] ];
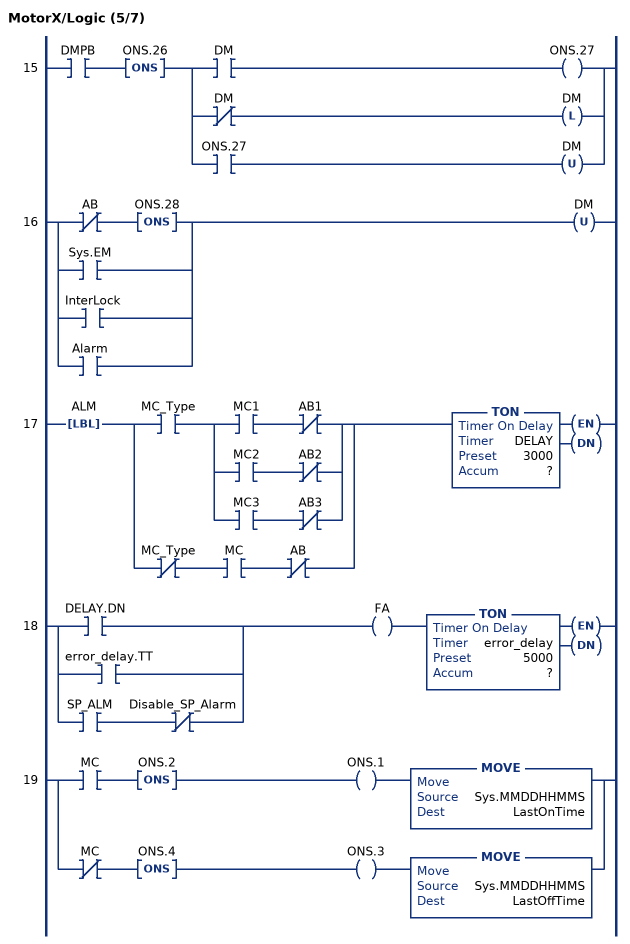
   15: XIC(DMPB)ONS(ONS.26)[XIC(DM) OTE(ONS.27) ,XIO(DM) OTL(DM) ,XIC(ONS.27) OTU(DM) ];
   16: [XIO(AB) ONS(ONS.28) ,XIC(Sys.EM) ,XIC(InterLock) ,XIC(Alarm) ]OTU(DM);
   17: LBL(ALM)[XIC(MC_Type) [XIC(MC1) XIO(AB1) ,XIC(MC2) XIO(AB2) ,XIC(MC3) XIO(AB3) ] ,XIO(MC_Type) XIC(MC) XIO(AB) ]TON(DELAY,?,?);
   18: [XIC(DELAY.DN) ,XIC(error_delay.TT) ,XIC(SP_ALM) XIO(Disable_SP_Alarm) ]OTE(FA)TON(error_delay,?,?);
   19: [XIC(MC) ONS(ONS.2) OTE(ONS.1) MOVE(Sys.MMDDHHMMS,LastOnTime) ,XIO(MC) ONS(ONS.4) OTE(ONS.3) MOVE(Sys.MMDDHHMMS,LastOffTime) ];
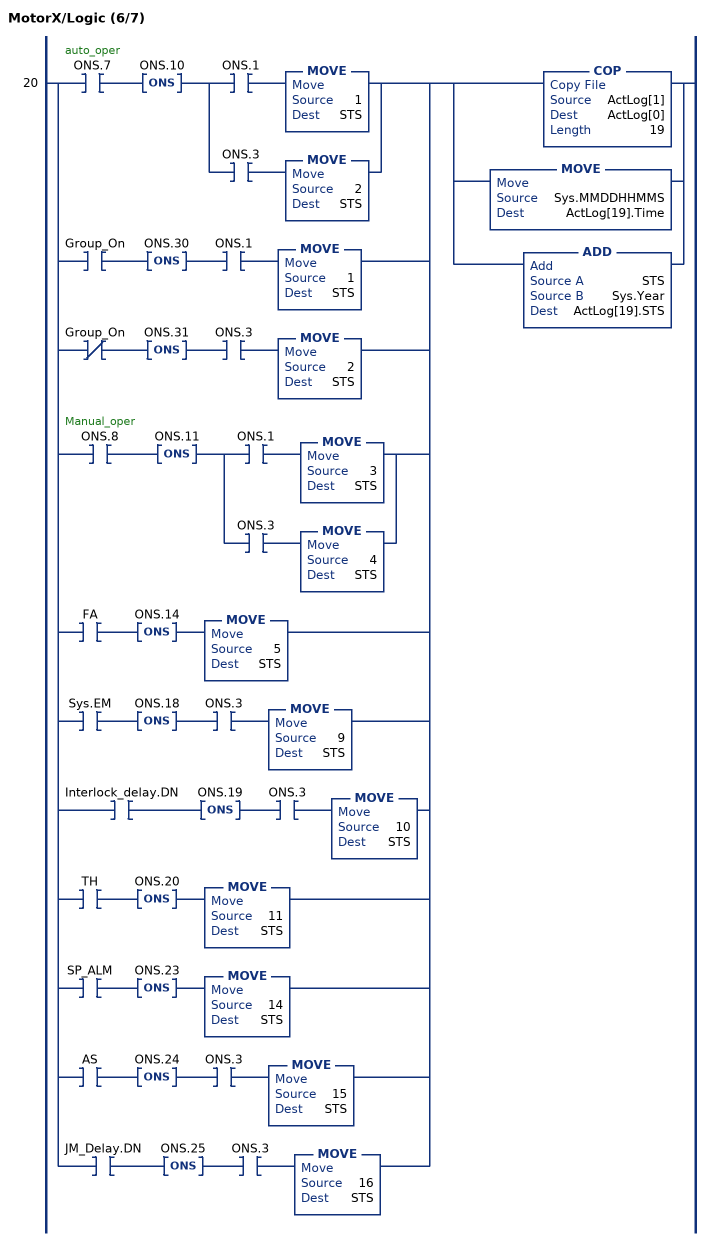
   20: [XIC(ONS.7) ONS(ONS.10) [XIC(ONS.1) MOVE(1,STS) ,XIC(ONS.3) MOVE(2,STS) ] ,XIC(Group_On) ONS(ONS.30) XIC(ONS.1) MOVE(1,STS) ,XIO(Group_On) ONS(ONS.31) XIC(ONS.3) MOVE(2,STS) ,XIC(ONS.8) ONS(ONS.11) [XIC(ONS.1) MOVE(3,STS) ,XIC(ONS.3) MOVE(4,STS) ] ,XIC(FA) ONS(ONS.14) MOVE(5,STS) ,XIC(Sys.EM) ONS(ONS.18) XIC(ONS.3) MOVE(9,STS) ,XIC(Interlock_delay.DN) ONS(ONS.19) XIC(ONS.3) MOVE(10,STS) ,XIC(TH) ONS(ONS.20) MOVE(11,STS) ,XIC(SP_ALM) ONS(ONS.23) MOVE(14,STS) ,XIC(AS) ONS(ONS.24) XIC(ONS.3) MOVE(15,STS) ,XIC(JM_Delay.DN) ONS(ONS.25) XIC(ONS.3) MOVE(16,STS) ][COP(ActLog[1],ActLog[0],19) ,MOVE(Sys.MMDDHHMMS,ActLog[19].Time) ,ADD(STS,Sys.Year,ActLog[19].STS) ];
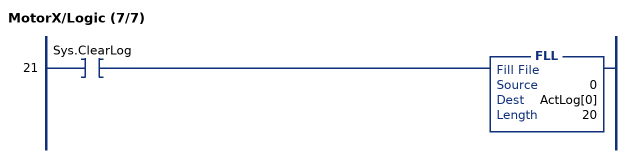
   21: XIC(Sys.ClearLog)FLL(0,ActLog[0],20);
END_ROUTINE
END_ADD_ON_INSTRUCTION
